ABB RobotStudio station: comportamiento2.rspag

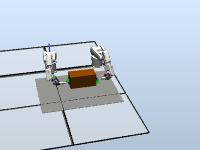
--- station ---
Station comportamiento2 (saved by RobotStudio 6.8.8307.1040)
Controller Sistema1, task T_ROB1: task frame (RAPID world) sits at (0, 807.58, 0) mm in the station
Controller IRB_120_3kg_0.58m
  mechanical unit ROB_1: IRB120_izda, 6 joints, base frame (0, 0, 0) mm
Controller Sistema1
  mechanical unit ROB_1: IRB120_dcha, 6 joints, base frame (0, 0, 0) mm
Layout (positions relative to the parent item):
  - IRB120_izda [mechanism, from Robots\IRB120_3_58_G_01.rslib] at (0, 0, 0) mm; joint values [-0.1452, 1.3679, -0.3747, 2.017, 1.2258, -1.0667] (rad or m)
  - MyTool_izda [mechanism, from Training Objects\myTool.rslib] at (529.1, -15.6, 125.16) mm, rotated rx 93.53 ry 0.68 rz 139.99 deg
  - IRB120_dcha [mechanism, from Robots\IRB120_3_58_G_01.rslib] at (0, 807.58, 0) mm; joint values [0.1851, 1.6156, -0.6679, -2.041, 1.4238, 1.2066] (rad or m)
  - MyTool_dcha [mechanism, from Training Objects\myTool.rslib] at (537.73, 843.66, 83.81) mm, rotated rx -81.65 ry 10.74 rz -140.82 deg
  - mesa [part] at (220.21, -292.83, 0) mm
  - caja [part] at (558.5, 202.06, 53.8) mm
  - Componente inteligente_1 [smart component]
      signals: DI coger
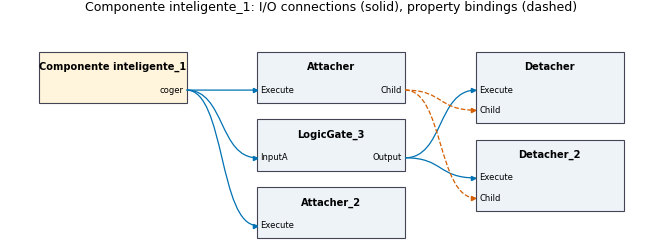
      connections:
        Componente inteligente_1.coger -> Attacher.Execute
        Componente inteligente_1.coger -> LogicGate_3.InputA
        LogicGate_3.Output -> Detacher.Execute
        Componente inteligente_1.coger -> Attacher_2.Execute
        LogicGate_3.Output -> Detacher_2.Execute
        Attacher.Child => Detacher.Child
        Attacher.Child => Detacher_2.Child
    - Detacher [smart component, from Components\Detacher.rslib]
        properties: Child=caja; KeepPosition=true
    - Attacher_2 [smart component, from Components\Attacher.rslib]
        properties: Parent=MyTool_dcha; Flange=0; Child=(none); Mount=false; Offset=[0 0 0]; Orientation=[0 0 0]
    - Attacher [smart component, from Components\Attacher.rslib]
        properties: Parent=MyTool_izda; Flange=0; Child=caja; Mount=false; Offset=[0 0 0]; Orientation=[0 0 0]
    - LogicGate_3 [smart component, from Components\LogicGate.rslib]
        properties: Operator=NOT; Delay=0
    - Detacher_2 [smart component, from Components\Detacher.rslib]
        properties: Child=caja; KeepPosition=true
  - LogicGate_4 [smart component, from Components\LogicGate.rslib]
      properties: Operator=AND; Delay=0
Attachment: MyTool_izda is attached to IRB120_izda / Link6
Attachment: MyTool_dcha is attached to IRB120_dcha / Link6
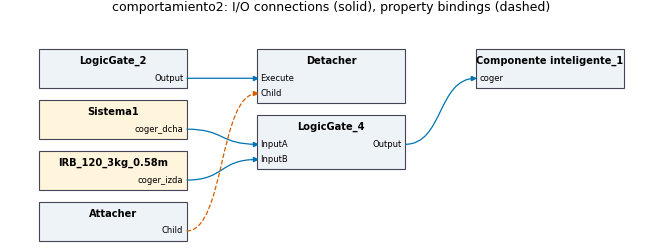
Station logic (signal -> signal, property => property):
  LogicGate_2.Output -> Detacher.Execute
  Sistema1.coger_dcha -> LogicGate_4.InputA
  IRB_120_3kg_0.58m.coger_izda -> LogicGate_4.InputB
  LogicGate_4.Output -> Componente inteligente_1.coger
  Attacher.Child => Detacher.Child

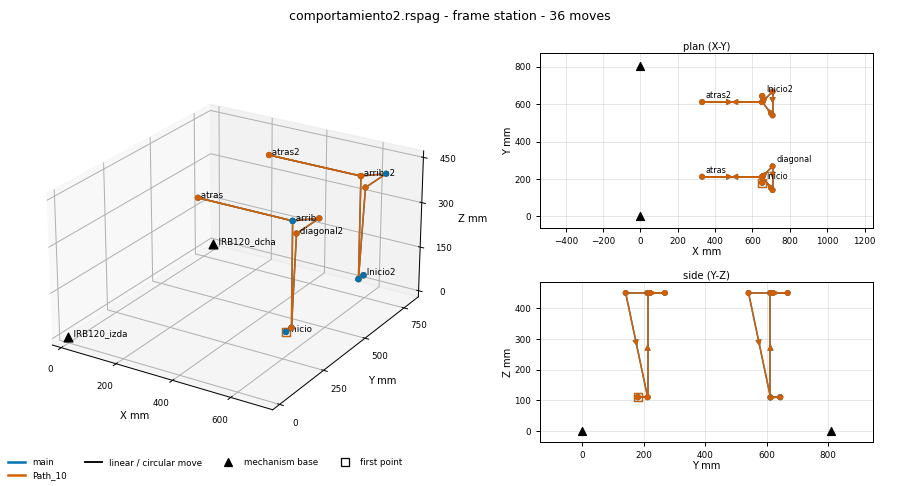
[picture p0: tool path of comportamiento2.rspag in frame station, 36 of 36 moves have a stored position in this frame; points joined in program order, loops and branches not executed]
--- Backups/IRB_120_3kg_0.58m/RAPID/TASK1/PROGMOD/CalibData.mod ---
MODULE CalibData
	PERS tooldata MyTool:=[TRUE,[[31.792631019,0,229.638935148],[0.945518576,0,0.325568154,0]],[1,[0,0,1],[1,0,0,0],0,0,0]];
ENDMODULE

--- Backups/IRB_120_3kg_0.58m/RAPID/TASK1/PROGMOD/Module1.mod ---
MODULE Module1
	CONST robtarget Inicio:=[[652.225,180.297,110.648],[0.002081155,0.022925495,0.72622909,0.687067246],[-1,1,-1,0],[9E+09,9E+09,9E+09,9E+09,9E+09,9E+09]];
	CONST robtarget Bloque1:=[[652.225,212.085,110.648],[0.002081155,0.022925495,0.72622909,0.687067246],[-1,1,-1,0],[9E+09,9E+09,9E+09,9E+09,9E+09,9E+09]];
	CONST robtarget arriba:=[[652.225,212.085,450.093],[0.002081155,0.022925495,0.72622909,0.687067246],[-1,1,-1,0],[9E+09,9E+09,9E+09,9E+09,9E+09,9E+09]];
	CONST robtarget atras:=[[330.24,212.085,450.093],[0.002081155,0.022925495,0.72622909,0.687067246],[-1,1,-1,0],[9E+09,9E+09,9E+09,9E+09,9E+09,9E+09]];
	CONST robtarget diagonal:=[[707.45810097,268.293908765,450.092991338],[0.002081065,0.022925358,0.726229084,0.687067257],[0,1,-1,0],[9E+09,9E+09,9E+09,9E+09,9E+09,9E+09]];
	CONST robtarget diagonal2:=[[707.458117808,140.673113523,450.092950644],[0.002080998,0.022925331,0.726229089,0.687067252],[-1,0,0,0],[9E+09,9E+09,9E+09,9E+09,9E+09,9E+09]];



    PROC main()
        !Path_10;
	    MoveL Inicio,v300,fine,MyTool\WObj:=wobj0;
	    MoveL Bloque1,v300,fine,MyTool\WObj:=wobj0;
        setdo coger_izda, 1;
	    MoveL arriba,v300,fine,MyTool\WObj:=wobj0;
	    MoveL atras,v300,fine,MyTool\WObj:=wobj0;
	    MoveL arriba,v300,fine,MyTool\WObj:=wobj0;
	    MoveL diagonal,v300,fine,MyTool\WObj:=wobj0;
	    MoveL diagonal2,v300,fine,MyTool\WObj:=wobj0;
	    MoveL Bloque1,v300,fine,MyTool\WObj:=wobj0;
        setdo coger_izda, 0;
	    MoveL Inicio,v300,fine,MyTool\WObj:=wobj0;

    ENDPROC


    PROC Path_10()
	    MoveL Inicio,v300,fine,MyTool\WObj:=wobj0;
	    MoveL Bloque1,v300,fine,MyTool\WObj:=wobj0;
	    MoveL arriba,v300,fine,MyTool\WObj:=wobj0;
	    MoveL atras,v300,fine,MyTool\WObj:=wobj0;
	    MoveL arriba,v300,fine,MyTool\WObj:=wobj0;
	    MoveL diagonal,v300,fine,MyTool\WObj:=wobj0;
	    MoveL diagonal2,v300,fine,MyTool\WObj:=wobj0;
	    MoveL Bloque1,v300,fine,MyTool\WObj:=wobj0;
	    MoveL Inicio,v300,fine,MyTool\WObj:=wobj0;
	ENDPROC
ENDMODULE

--- Backups/Sistema1/RAPID/TASK1/PROGMOD/Module1.mod ---
MODULE Module1
	CONST robtarget Inicio2:=[[652.224,-163.703473649,110.648],[0.085920466,0.081141772,0.70324444,-0.701057019],[0,-2,0,0],[9E+09,9E+09,9E+09,9E+09,9E+09,9E+09]];
	CONST robtarget Bloque2:=[[652.224,-195.491473649,110.058],[0.085920466,0.081141772,0.70324444,-0.701057019],[0,-2,0,0],[9E+09,9E+09,9E+09,9E+09,9E+09,9E+09]];
	CONST robtarget arriba2:=[[652.224,-195.491473649,450.093],[0.085920466,0.081141772,0.70324444,-0.701057019],[0,-2,0,0],[9E+09,9E+09,9E+09,9E+09,9E+09,9E+09]];
	CONST robtarget atras2:=[[330.24,-195.491473649,450.093],[0.085920466,0.081141772,0.70324444,-0.701057019],[0,-2,0,0],[9E+09,9E+09,9E+09,9E+09,9E+09,9E+09]];
	CONST robtarget diagonal:=[[707.456981771,-139.282718953,450.092981236],[0.085920454,0.081141778,0.703244402,-0.701057058],[0,-2,0,0],[9E+09,9E+09,9E+09,9E+09,9E+09,9E+09]];
	CONST robtarget diagonal2:=[[707.457031068,-266.903615707,450.092932882],[0.085920438,0.081141753,0.703244366,-0.701057099],[-1,-2,0,0],[9E+09,9E+09,9E+09,9E+09,9E+09,9E+09]];

    PROC main()
        !Path_10;
	    MoveL Inicio2,v300,fine,MyTool\WObj:=wobj0;
	    MoveL Bloque2,v300,fine,MyTool\WObj:=wobj0;
	    SetDO coger_dcha, 1;
        MoveL arriba2,v300,fine,MyTool\WObj:=wobj0;
	    MoveL atras2,v300,fine,MyTool\WObj:=wobj0;
	    MoveL arriba2,v300,fine,MyTool\WObj:=wobj0;
	    MoveL diagonal,v300,fine,MyTool\WObj:=wobj0;
	    MoveL diagonal2,v300,fine,MyTool\WObj:=wobj0;
	    MoveL Bloque2,v300,fine,MyTool\WObj:=wobj0;
	    SetDo coger_dcha, 0;
        MoveL Inicio2,v300,fine,MyTool\WObj:=wobj0;
    ENDPROC

    PROC Path_10()
	    MoveL Inicio2,v300,fine,MyTool\WObj:=wobj0;
	    MoveL Bloque2,v300,fine,MyTool\WObj:=wobj0;
	    MoveL arriba2,v300,fine,MyTool\WObj:=wobj0;
	    MoveL atras2,v300,fine,MyTool\WObj:=wobj0;
	    MoveL arriba2,v300,fine,MyTool\WObj:=wobj0;
	    MoveL diagonal,v300,fine,MyTool\WObj:=wobj0;
	    MoveL diagonal2,v300,fine,MyTool\WObj:=wobj0;
	    MoveL Bloque2,v300,fine,MyTool\WObj:=wobj0;
	    MoveL Inicio2,v300,fine,MyTool\WObj:=wobj0;
	ENDPROC
ENDMODULE

--- Backups/IRB_120_3kg_0.58m/SYSPAR/EIO.cfg ---
EIO:CFG_1.0:6:1::
#
EIO_SIGNAL:

      -Name "coger_izda" -SignalType "DO"

--- Backups/Sistema1/SYSPAR/EIO.cfg ---
EIO:CFG_1.0:6:1::
#
EIO_SIGNAL:

      -Name "coger_dcha" -SignalType "DO"
